# B&R Automation Studio project PO-Laba2
Automation Studio 4.5.2.102

## Logical view

Binary libraries used (declarations not repeated): operator, runtime, astime, AsIecCon, Acp10par, NcGlobal, Acp10man, Acp10sdc, Acp10_MC, brsystem, sys_lib, AsBrStr

### Library Logical/Libraries/DriveLib (ANSIC)

#### Types.typ
```iecst
TYPE
	CmddCodes :
		(
		CMD_SHUTDOWN := 6,
		CMD_SWITCH_ON := 7,
		CMD_ENABLED := 15
		);
	DoorStates :
		(
		ST_INIT,
		ST_UNKNOWN,
		ST_OPEN,
		ST_CLOSE,
		ST_ACC_POS,
		ST_ACC_NEG,
		ST_POS,
		ST_NEG,
		ST_DEC_POS,
		ST_DEC_NEG
		);
	EtadCodes :
		(
		STATE_DISABLED := 64,
		STATE_SWITCH_ON := 35,
		STATE_READY := 33
		);
END_TYPE
```

#### DriveLib.fun
```iecst
{REDUND_ERROR} FUNCTION_BLOCK FB_DoorSM (*TODO: Add your comment here*) (*$GROUP=User,$CAT=User,$GROUPICON=User.png,$CATICON=User.png*)
	VAR_INPUT
		state : UINT;
		sw1 : BOOL;
		sw2 : BOOL;
		sw3 : BOOL;
		sw4 : BOOL;
		direction : BOOL;
	END_VAR
	VAR_OUTPUT
		speed : INT;
	END_VAR
	VAR
		swo1 : BOOL;
		swo2 : BOOL;
		swo3 : BOOL;
		swo4 : BOOL;
	END_VAR
END_FUNCTION_BLOCK

{REDUND_ERROR} FUNCTION_BLOCK FB_LedSM (*TODO: Add your comment here*) (*$GROUP=User,$CAT=User,$GROUPICON=User.png,$CATICON=User.png*)
	VAR_INPUT
		state : UINT;
	END_VAR
	VAR_OUTPUT
		led1 : BOOL;
		led2 : BOOL;
		led3 : BOOL;
		led4 : BOOL;
		timer : INT;
	END_VAR
END_FUNCTION_BLOCK

{REDUND_ERROR} FUNCTION_BLOCK FB_StateMachine (*TODO: Add your comment here*) (*$GROUP=User,$CAT=User,$GROUPICON=User.png,$CATICON=User.png*)
	VAR_INPUT
		state : UINT;
		enable : BOOL;
	END_VAR
	VAR_OUTPUT
		command : UINT;
		speed : INT;
	END_VAR
END_FUNCTION_BLOCK
```

#### FB_DoorSM.c
```c
#include <bur/plctypes.h>
#ifdef __cplusplus
	extern "C"
	{
#endif
	#include "DriveLib.h"
#ifdef __cplusplus
	};
#endif
/* TODO: Add your comment here */
void FB_DoorSM(struct FB_DoorSM* inst)
{
    switch (inst->state) {
        case ST_INIT:
			if (inst->sw1==0 && inst->sw2==0 && inst->sw3==0 && inst->sw4==0) {
				inst->state=ST_UNKNOWN;
			}
            break;
        case ST_UNKNOWN:
            if (inst->direction == 0 && inst->sw1!=inst->swo1) {
                inst->state = ST_OPEN;
            }
            if (inst->direction == 0 && inst->sw2!=inst->swo2) {
                inst->state = ST_ACC_NEG;
            }
            if (inst->direction == 0 && inst->sw3!=inst->swo3) {
                inst->state = ST_NEG;
            }
            if (inst->direction == 0 && inst->sw4!=inst->swo4) {
                inst->state = ST_DEC_NEG;
            }
            if (inst->direction == 1 && inst->sw4!=inst->swo4) {
                inst->state = ST_CLOSE;
            }
            if (inst->direction == 1 && inst->sw3!=inst->swo3) {
                inst->state = ST_ACC_POS;
            }
            if (inst->direction == 1 && inst->sw2!=inst->swo2) {
                inst->state = ST_POS;
            }
            if (inst->direction == 1 && inst->sw1!=inst->swo1) {
                inst->state = ST_DEC_POS;
            }
            break;
        case ST_OPEN:
            inst->speed=0;
            if (inst->direction == 0) {
                inst->state = ST_ACC_NEG;
            }
            break;
        case ST_ACC_NEG:
            inst->speed=250;
            if (inst->direction == 0 && inst->sw2!=inst->swo2) {
                inst->state = ST_NEG;
            }
            if (inst->direction == 1) {
                inst->state = ST_DEC_NEG;
            }
            break;
        case ST_NEG:
            inst->speed=800;
			if (inst->direction == 0 && inst->sw3!=inst->swo3) {
                inst->state = ST_DEC_NEG;
            }
            if (inst->direction == 1) {
                inst->state = ST_POS;
            }
            break;
        case ST_DEC_NEG:
            inst->speed=250;
            if (inst->sw4 == !inst->swo4) {
                inst->state = ST_CLOSE;
            }
            break;
        case ST_CLOSE:
            inst->speed=0;
            if (inst->direction == 1) {
                inst->state = ST_ACC_POS;
            }
            break;
		case ST_ACC_POS:
			inst->speed=-250;
            if (inst->direction == 1 && inst->sw3!=inst->swo3) {
                inst->state = ST_POS;
            }
            if (inst->direction == 0) {
                inst->state = ST_DEC_POS;
            }
            break;
        case ST_POS:
            inst->speed=-800;
            if (inst->direction == 1 && inst->sw2!=inst->swo2) {
                inst->state = ST_DEC_POS;
            }
            if (inst->direction == 0) {
                inst->state = ST_NEG;
            }
            break;
		case ST_DEC_POS:
			inst->speed=-250;
            if (inst->sw1!=inst->swo1) {
                inst->state = ST_OPEN;
            }
            break;
    }

    inst->swo1=inst->sw1;
    inst->swo2=inst->sw2;
    inst->swo3=inst->sw3;
    inst->swo4=inst->sw4;
}
```

#### FB_LedSM.c
```c
#include <bur/plctypes.h>
#ifdef __cplusplus
	extern "C"
	{
#endif
	#include "DriveLib.h"
#ifdef __cplusplus
	};
#endif
/* TODO: Add your comment here */
void FB_LedSM(struct FB_LedSM* inst)
{
    switch(inst->state) {
        case ST_INIT:
            break;
        case ST_UNKNOWN:
            if (inst->timer%11==10)
                inst->led1 = !inst->led1;
                inst->led2 = !inst->led2;
                inst->led3 = !inst->led3;
                inst->led4 = !inst->led4;
            break;
        case ST_OPEN:
            inst->led1 = 0;
            inst->led2 = 0;
            inst->led3 = 0;
            inst->led4 = 0;
            break;
        case ST_ACC_NEG:
			inst->led1 = 1;
			if (inst->timer%21==20)
				inst->led2 = !inst->led2;
            inst->led3 = 0;
            inst->led4 = 0;
            break;
        case ST_NEG:
            inst->led1 = 1;
			inst->led2 = 1;
			if (inst->timer%11==10)
				inst->led3 = !inst->led3;
            inst->led4 = 0;
            break;
        case ST_DEC_NEG:
            inst->led1 = 1;
            inst->led2 = 1;
			inst->led3 = 1;
			if (inst->timer%21==20)
				inst->led4 = !inst->led4;
            break;
        case ST_CLOSE:
            inst->led1 = 1;
            inst->led2 = 1;
            inst->led3 = 1;
            inst->led4 = 1;
            break;
        case ST_ACC_POS:
            inst->led1 = 1;
			inst->led2 = 1;
			if (inst->timer%21==20)
				inst->led3 = !inst->led3;
            inst->led4 = 0;
            break;
        case ST_POS:
			inst->led1 = 1;
			if (inst->timer%11==10)
				inst->led2 = !inst->led2;
            inst->led3 = 0;
            inst->led4 = 0;
            break;
		case ST_DEC_POS:
			if (inst->timer%21==20)
				inst->led1 = !inst->led1;
            inst->led2 = 0;
            inst->led3 = 0;
            inst->led4 = 0;
            break;
    }
    inst->timer++;
}
```

### Library Logical/Library (ANSIC)

#### Library.fun
```iecst
{REDUND_ERROR} FUNCTION_BLOCK stateMachine (*TODO: Add your comment here*) (*$GROUP=User,$CAT=User,$GROUPICON=User.png,$CATICON=User.png*)
	VAR_INPUT
		state : UINT;
		enable : BOOL;
	END_VAR
	VAR_OUTPUT
		command : UINT;
		speed : INT;
	END_VAR
END_FUNCTION_BLOCK

{REDUND_ERROR} FUNCTION_BLOCK doorSM (*TODO: Add your comment here*) (*$GROUP=User,$CAT=User,$GROUPICON=User.png,$CATICON=User.png*)
	VAR_INPUT
		state : BOOL;
		sw1 : BOOL;
		sw2 : BOOL;
		sw3 : BOOL;
		sw4 : BOOL;
		direction : BOOL;
	END_VAR
	VAR_OUTPUT
		speed : INT;
	END_VAR
END_FUNCTION_BLOCK

{REDUND_ERROR} FUNCTION_BLOCK ledSM (*TODO: Add your comment here*) (*$GROUP=User,$CAT=User,$GROUPICON=User.png,$CATICON=User.png*)
	VAR_INPUT
		state : BOOL;
		led1 : BOOL;
		led2 : BOOL;
		led3 : BOOL;
		led4 : BOOL;
	END_VAR
	VAR_OUTPUT
		timer : INT;
	END_VAR
END_FUNCTION_BLOCK
```

#### stateMachine.c
```c
#include <bur/plctypes.h>
#ifdef __cplusplus
	extern "C"
	{
#endif
	#include "Library.h"
#ifdef __cplusplus
	};
#endif
/* TODO: Add your comment here */
void stateMachine(struct stateMachine* inst)
{
	/*TODO: Add your code here*/
}
```

#### doorSM.c
```c
#include <bur/plctypes.h>
#ifdef __cplusplus
	extern "C"
	{
#endif
	#include "Library.h"
#ifdef __cplusplus
	};
#endif
/* TODO: Add your comment here */
void doorSM(struct doorSM* inst)
{
	/*TODO: Add your code here*/
}
```

#### ledSM.c
```c
#include <bur/plctypes.h>
#ifdef __cplusplus
	extern "C"
	{
#endif
	#include "Library.h"
#ifdef __cplusplus
	};
#endif
/* TODO: Add your comment here */
void ledSM(struct ledSM* inst)
{
	/*TODO: Add your code here*/
}
```

Listed in the project but not available here: Logical/Library/Types.typ, Logical/Library/Constants.var
